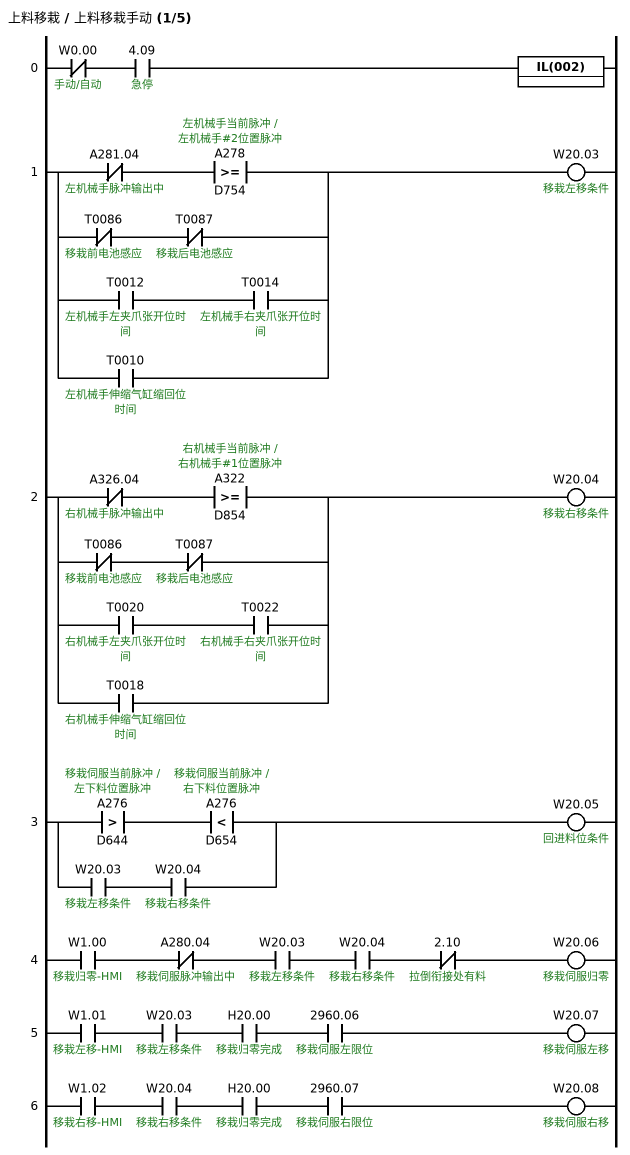
; [picture p89: 上料移栽 / 上料移栽手动, rungs 0-6]
; rung 0
LDNOT W0.00  ; 手动/自动
AND 4.09  ; 急停
IL(002)
; rung 1
LDNOT A281.04  ; 左机械手脉冲输出中
AND>=SL(328) A278 D754  ; 左机械手当前脉冲, 左机械手#2位置脉冲
LDNOT T0086  ; 移栽前电池感应
ANDNOT T0087  ; 移栽后电池感应
ORLD
LD T0012  ; 左机械手左夹爪张开位时间
AND T0014  ; 左机械手右夹爪张开位时间
ORLD
OR T0010  ; 左机械手伸缩气缸缩回位时间
OUT W20.03  ; 移栽左移条件
; rung 2
LDNOT A326.04  ; 右机械手脉冲输出中
AND>=SL(328) A322 D854  ; 右机械手当前脉冲, 右机械手#1位置脉冲
LDNOT T0086  ; 移栽前电池感应
ANDNOT T0087  ; 移栽后电池感应
ORLD
LD T0020  ; 右机械手左夹爪张开位时间
AND T0022  ; 右机械手右夹爪张开位时间
ORLD
OR T0018  ; 右机械手伸缩气缸缩回位时间
OUT W20.04  ; 移栽右移条件
; rung 3
LD>SL(323) A276 D644  ; 移栽伺服当前脉冲, 左下料位置脉冲
AND<SL(313) A276 D654  ; 移栽伺服当前脉冲, 右下料位置脉冲
LD W20.03  ; 移栽左移条件
AND W20.04  ; 移栽右移条件
ORLD
OUT W20.05  ; 回进料位条件
; rung 4
LD W1.00  ; 移栽归零-HMI
ANDNOT A280.04  ; 移栽伺服脉冲输出中
AND W20.03  ; 移栽左移条件
AND W20.04  ; 移栽右移条件
ANDNOT 2.10  ; 拉倒衔接处有料
OUT W20.06  ; 移栽伺服归零
; rung 5
LD W1.01  ; 移栽左移-HMI
AND W20.03  ; 移栽左移条件
AND H20.00  ; 移栽归零完成
AND 2960.06  ; 移栽伺服左限位
OUT W20.07  ; 移栽伺服左移
; rung 6
LD W1.02  ; 移栽右移-HMI
AND W20.04  ; 移栽右移条件
AND H20.00  ; 移栽归零完成
AND 2960.07  ; 移栽伺服右限位
OUT W20.08  ; 移栽伺服右移

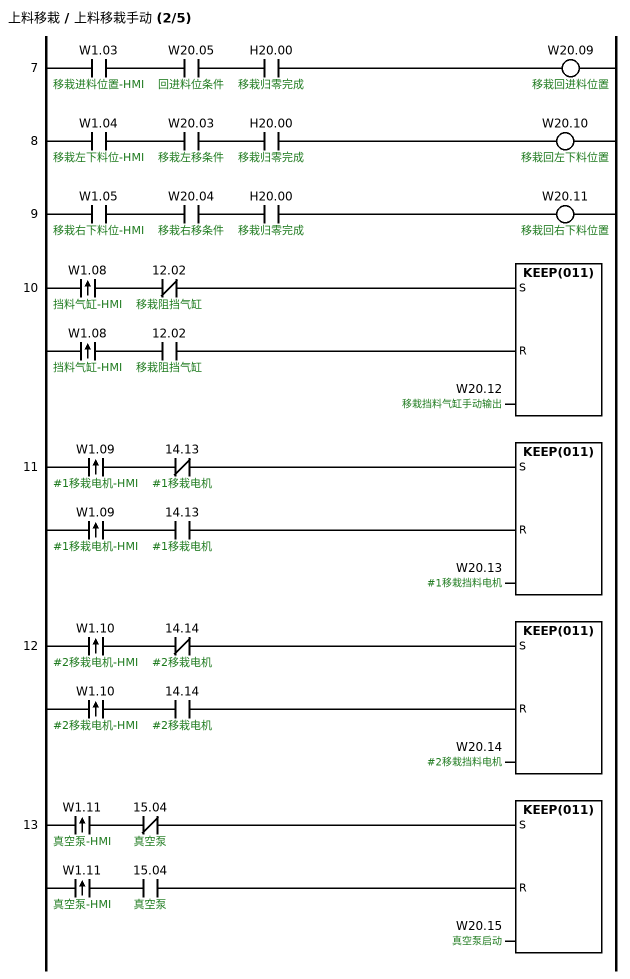
; rung 7
LD W1.03  ; 移栽进料位置-HMI
AND W20.05  ; 回进料位条件
AND H20.00  ; 移栽归零完成
OUT W20.09  ; 移栽回进料位置
; rung 8
LD W1.04  ; 移栽左下料位-HMI
AND W20.03  ; 移栽左移条件
AND H20.00  ; 移栽归零完成
OUT W20.10  ; 移栽回左下料位置
; rung 9
LD W1.05  ; 移栽右下料位-HMI
AND W20.04  ; 移栽右移条件
AND H20.00  ; 移栽归零完成
OUT W20.11  ; 移栽回右下料位置
; rung 10
@LD W1.08  ; 挡料气缸-HMI
ANDNOT 12.02  ; 移栽阻挡气缸
@LD W1.08  ; 挡料气缸-HMI
AND 12.02  ; 移栽阻挡气缸
KEEP(011) W20.12  ; 移栽挡料气缸手动输出
; rung 11
@LD W1.09  ; #1移栽电机-HMI
ANDNOT 14.13  ; #1移栽电机
@LD W1.09  ; #1移栽电机-HMI
AND 14.13  ; #1移栽电机
KEEP(011) W20.13  ; #1移栽挡料电机
; rung 12
@LD W1.10  ; #2移栽电机-HMI
ANDNOT 14.14  ; #2移栽电机
@LD W1.10  ; #2移栽电机-HMI
AND 14.14  ; #2移栽电机
KEEP(011) W20.14  ; #2移栽挡料电机
; rung 13
@LD W1.11  ; 真空泵-HMI
ANDNOT 15.04  ; 真空泵
@LD W1.11  ; 真空泵-HMI
AND 15.04  ; 真空泵
KEEP(011) W20.15  ; 真空泵启动

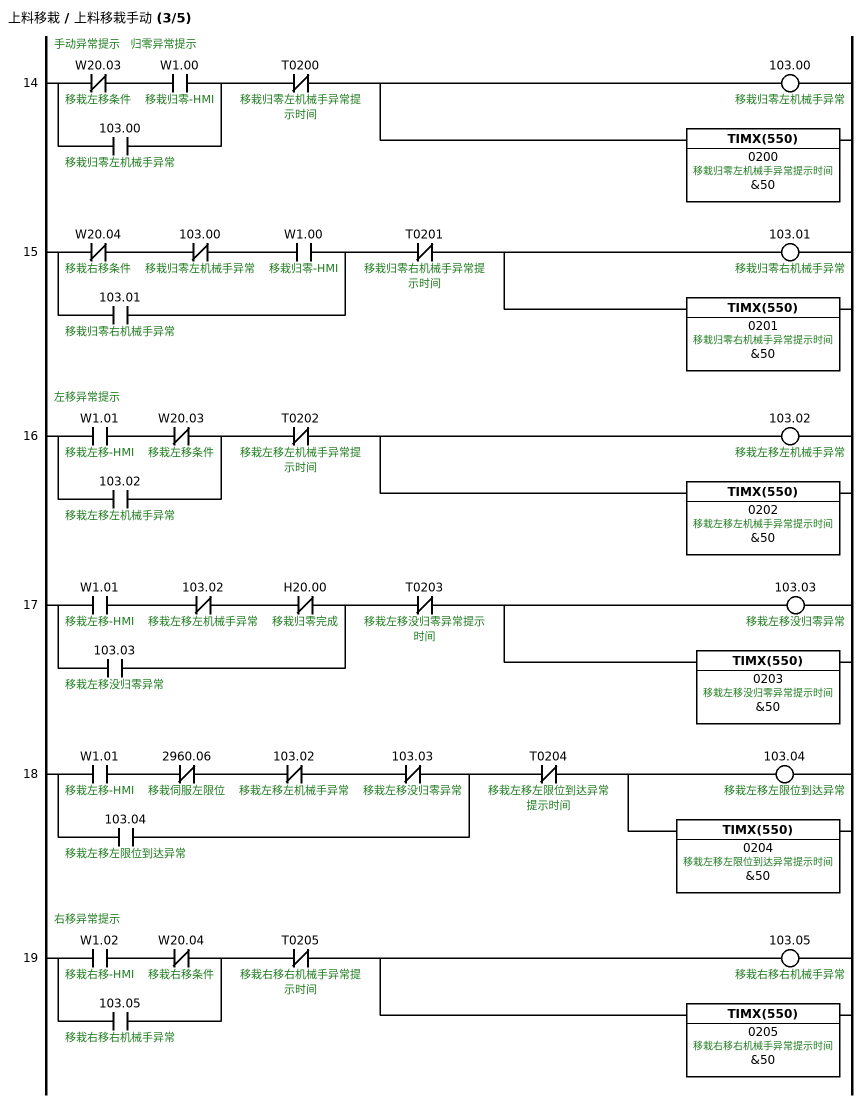
; rung 14: 手动异常提示   归零异常提示
LDNOT W20.03  ; 移栽左移条件
AND W1.00  ; 移栽归零-HMI
OR 103.00  ; 移栽归零左机械手异常
ANDNOT T0200  ; 移栽归零左机械手异常提示时间
OUT 103.00  ; 移栽归零左机械手异常
TIMX(550) 0200 &50  ; 移栽归零左机械手异常提示时间
; rung 15
LDNOT W20.04  ; 移栽右移条件
ANDNOT 103.00  ; 移栽归零左机械手异常
AND W1.00  ; 移栽归零-HMI
OR 103.01  ; 移栽归零右机械手异常
ANDNOT T0201  ; 移栽归零右机械手异常提示时间
OUT 103.01  ; 移栽归零右机械手异常
TIMX(550) 0201 &50  ; 移栽归零右机械手异常提示时间
; rung 16: 左移异常提示
LD W1.01  ; 移栽左移-HMI
ANDNOT W20.03  ; 移栽左移条件
OR 103.02  ; 移栽左移左机械手异常
ANDNOT T0202  ; 移栽左移左机械手异常提示时间
OUT 103.02  ; 移栽左移左机械手异常
TIMX(550) 0202 &50  ; 移栽左移左机械手异常提示时间
; rung 17
LD W1.01  ; 移栽左移-HMI
ANDNOT 103.02  ; 移栽左移左机械手异常
ANDNOT H20.00  ; 移栽归零完成
OR 103.03  ; 移栽左移没归零异常
ANDNOT T0203  ; 移栽左移没归零异常提示时间
OUT 103.03  ; 移栽左移没归零异常
TIMX(550) 0203 &50  ; 移栽左移没归零异常提示时间
; rung 18
LD W1.01  ; 移栽左移-HMI
ANDNOT 2960.06  ; 移栽伺服左限位
ANDNOT 103.02  ; 移栽左移左机械手异常
ANDNOT 103.03  ; 移栽左移没归零异常
OR 103.04  ; 移栽左移左限位到达异常
ANDNOT T0204  ; 移栽左移左限位到达异常提示时间
OUT 103.04  ; 移栽左移左限位到达异常
TIMX(550) 0204 &50  ; 移栽左移左限位到达异常提示时间
; rung 19: 右移异常提示
LD W1.02  ; 移栽右移-HMI
ANDNOT W20.04  ; 移栽右移条件
OR 103.05  ; 移栽右移右机械手异常
ANDNOT T0205  ; 移栽右移右机械手异常提示时间
OUT 103.05  ; 移栽右移右机械手异常
TIMX(550) 0205 &50  ; 移栽右移右机械手异常提示时间

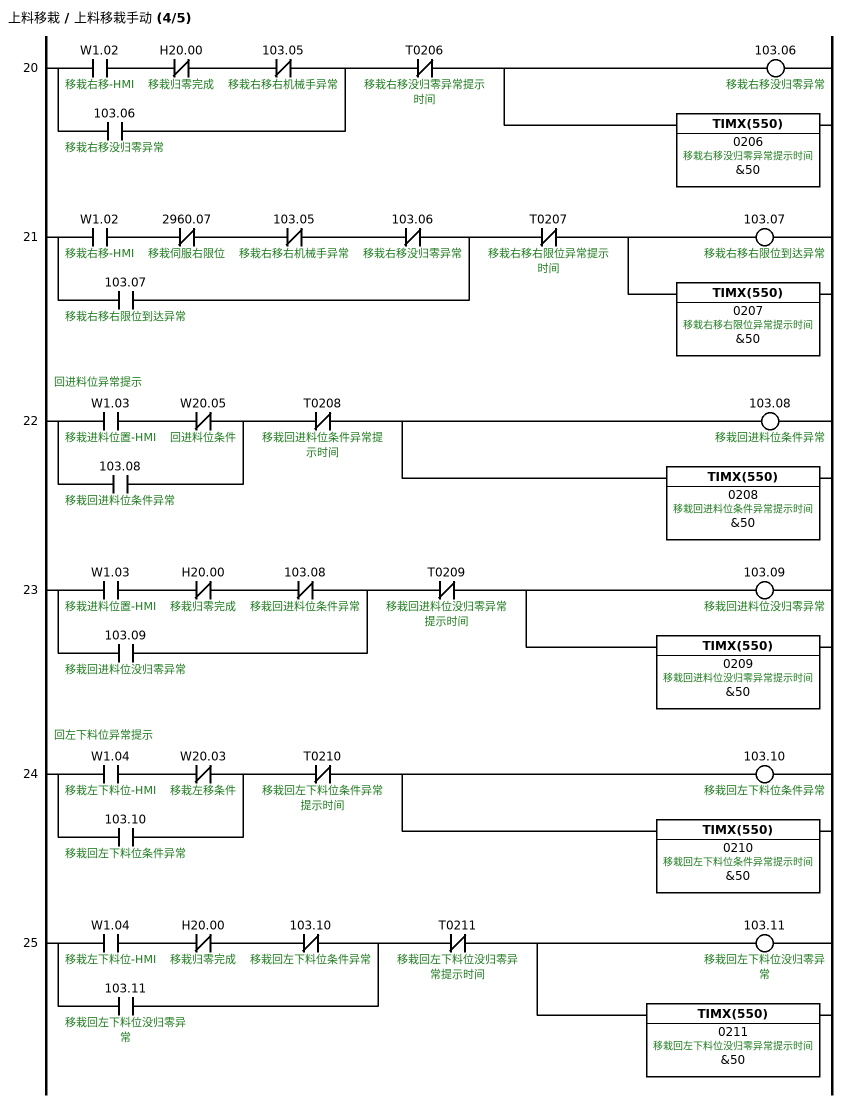
; rung 20
LD W1.02  ; 移栽右移-HMI
ANDNOT H20.00  ; 移栽归零完成
ANDNOT 103.05  ; 移栽右移右机械手异常
OR 103.06  ; 移栽右移没归零异常
ANDNOT T0206  ; 移栽右移没归零异常提示时间
OUT 103.06  ; 移栽右移没归零异常
TIMX(550) 0206 &50  ; 移栽右移没归零异常提示时间
; rung 21
LD W1.02  ; 移栽右移-HMI
ANDNOT 2960.07  ; 移栽伺服右限位
ANDNOT 103.05  ; 移栽右移右机械手异常
ANDNOT 103.06  ; 移栽右移没归零异常
OR 103.07  ; 移栽右移右限位到达异常
ANDNOT T0207  ; 移栽右移右限位异常提示时间
OUT 103.07  ; 移栽右移右限位到达异常
TIMX(550) 0207 &50  ; 移栽右移右限位异常提示时间
; rung 22: 回进料位异常提示
LD W1.03  ; 移栽进料位置-HMI
ANDNOT W20.05  ; 回进料位条件
OR 103.08  ; 移栽回进料位条件异常
ANDNOT T0208  ; 移栽回进料位条件异常提示时间
OUT 103.08  ; 移栽回进料位条件异常
TIMX(550) 0208 &50  ; 移栽回进料位条件异常提示时间
; rung 23
LD W1.03  ; 移栽进料位置-HMI
ANDNOT H20.00  ; 移栽归零完成
ANDNOT 103.08  ; 移栽回进料位条件异常
OR 103.09  ; 移栽回进料位没归零异常
ANDNOT T0209  ; 移栽回进料位没归零异常提示时间
OUT 103.09  ; 移栽回进料位没归零异常
TIMX(550) 0209 &50  ; 移栽回进料位没归零异常提示时间
; rung 24: 回左下料位异常提示
LD W1.04  ; 移栽左下料位-HMI
ANDNOT W20.03  ; 移栽左移条件
OR 103.10  ; 移栽回左下料位条件异常
ANDNOT T0210  ; 移栽回左下料位条件异常提示时间
OUT 103.10  ; 移栽回左下料位条件异常
TIMX(550) 0210 &50  ; 移栽回左下料位条件异常提示时间
; rung 25
LD W1.04  ; 移栽左下料位-HMI
ANDNOT H20.00  ; 移栽归零完成
ANDNOT 103.10  ; 移栽回左下料位条件异常
OR 103.11  ; 移栽回左下料位没归零异常
ANDNOT T0211  ; 移栽回左下料位没归零异常提示时间
OUT 103.11  ; 移栽回左下料位没归零异常
TIMX(550) 0211 &50  ; 移栽回左下料位没归零异常提示时间

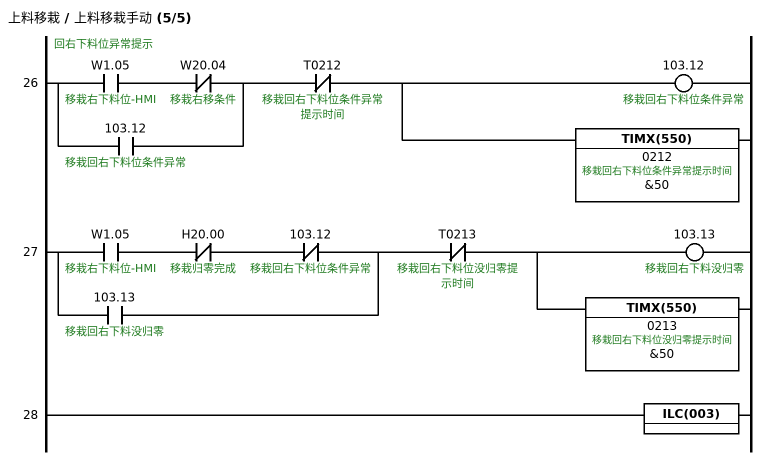
; rung 26: 回右下料位异常提示
LD W1.05  ; 移栽右下料位-HMI
ANDNOT W20.04  ; 移栽右移条件
OR 103.12  ; 移栽回右下料位条件异常
ANDNOT T0212  ; 移栽回右下料位条件异常提示时间
OUT 103.12  ; 移栽回右下料位条件异常
TIMX(550) 0212 &50  ; 移栽回右下料位条件异常提示时间
; rung 27
LD W1.05  ; 移栽右下料位-HMI
ANDNOT H20.00  ; 移栽归零完成
ANDNOT 103.12  ; 移栽回右下料位条件异常
OR 103.13  ; 移栽回右下料没归零
ANDNOT T0213  ; 移栽回右下料位没归零提示时间
OUT 103.13  ; 移栽回右下料没归零
TIMX(550) 0213 &50  ; 移栽回右下料位没归零提示时间
; rung 28
ILC(003)

### Section 上料移栽自动

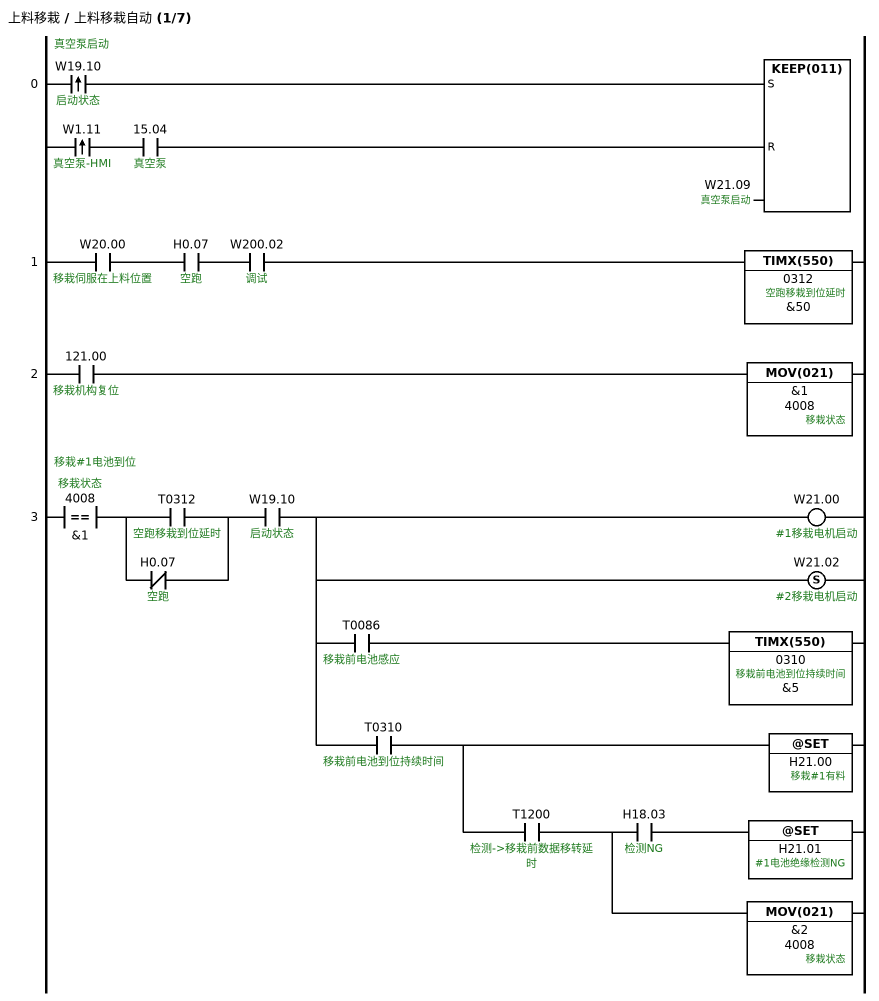
; rung 0: 真空泵启动
@LD W19.10  ; 启动状态
@LD W1.11  ; 真空泵-HMI
AND 15.04  ; 真空泵
KEEP(011) W21.09  ; 真空泵启动
; rung 1
LD W20.00  ; 移栽伺服在上料位置
AND H0.07  ; 空跑
AND W200.02  ; 调试
TIMX(550) 0312 &50  ; 空跑移栽到位延时
; rung 2
LD 121.00  ; 移栽机构复位
MOV(021) &1 4008  ; 移栽状态
; rung 3: 移栽#1电池到位
LD=(300) 4008 &1  ; 移栽状态
LD T0312  ; 空跑移栽到位延时
ORNOT H0.07  ; 空跑
ANDLD
AND W19.10  ; 启动状态
OUT TR0
OUT W21.00  ; #1移栽电机启动
SET W21.02  ; #2移栽电机启动
AND T0086  ; 移栽前电池感应
TIMX(550) 0310 &5  ; 移栽前电池到位持续时间
LD TR0
AND T0310  ; 移栽前电池到位持续时间
@SET H21.00  ; 移栽#1有料
AND T1200  ; 检测->移栽前数据移转延时
OUT TR0
AND H18.03  ; 检测NG
@SET H21.01  ; #1电池绝缘检测NG
LD TR0
MOV(021) &2 4008  ; 移栽状态

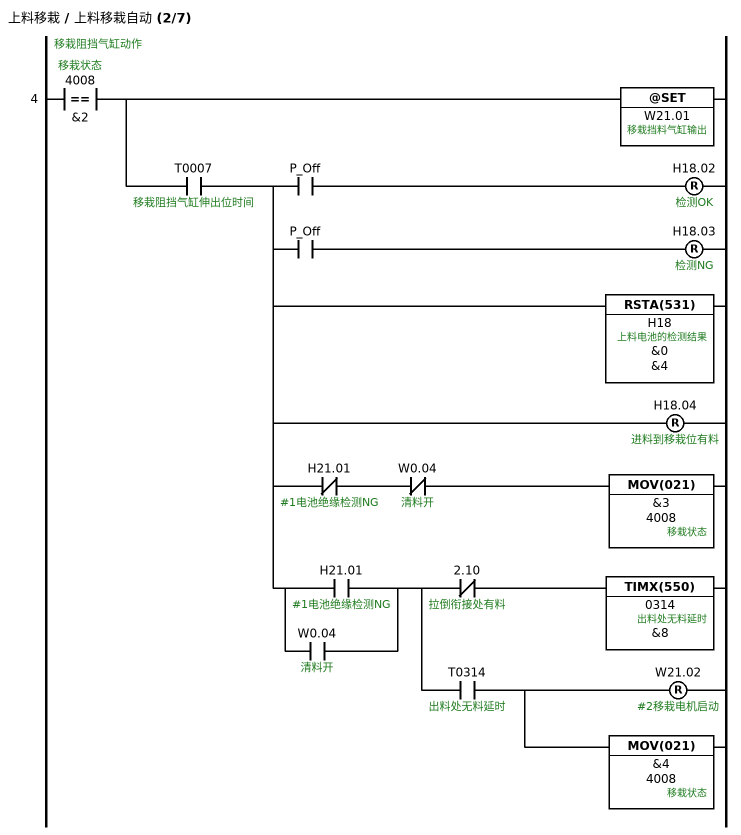
; rung 4: 移栽阻挡气缸动作
LD=(300) 4008 &2  ; 移栽状态
@SET W21.01  ; 移栽挡料气缸输出
AND T0007  ; 移栽阻挡气缸伸出位时间
OUT TR0
AND P_Off
RSET H18.02  ; 检测OK
LD TR0
AND P_Off
RSET H18.03  ; 检测NG
LD TR0
RSTA(531) H18 &0 &4  ; 上料电池的检测结果
RSET H18.04  ; 进料到移栽位有料
ANDNOT H21.01  ; #1电池绝缘检测NG
ANDNOT W0.04  ; 清料开
MOV(021) &3 4008  ; 移栽状态
LD TR0
LD H21.01  ; #1电池绝缘检测NG
OR W0.04  ; 清料开
ANDLD
OUT TR0
ANDNOT 2.10  ; 拉倒衔接处有料
TIMX(550) 0314 &8  ; 出料处无料延时
LD TR0
AND T0314  ; 出料处无料延时
RSET W21.02  ; #2移栽电机启动
MOV(021) &4 4008  ; 移栽状态

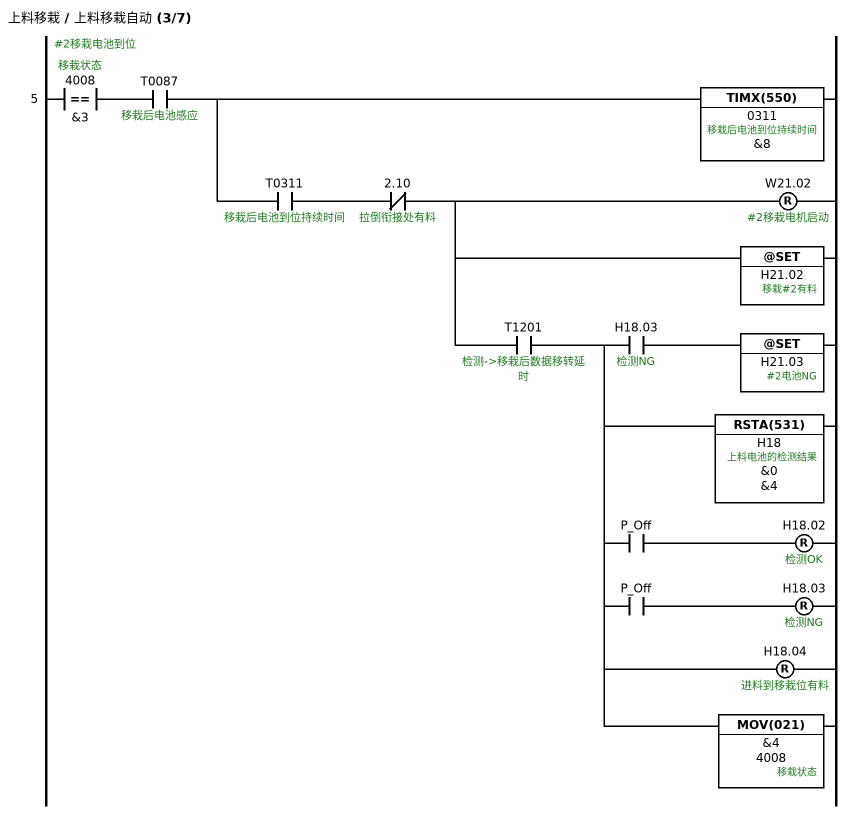
; rung 5: #2移栽电池到位
LD=(300) 4008 &3  ; 移栽状态
AND T0087  ; 移栽后电池感应
TIMX(550) 0311 &8  ; 移栽后电池到位持续时间
AND T0311  ; 移栽后电池到位持续时间
ANDNOT 2.10  ; 拉倒衔接处有料
RSET W21.02  ; #2移栽电机启动
@SET H21.02  ; 移栽#2有料
AND T1201  ; 检测->移栽后数据移转延时
OUT TR0
AND H18.03  ; 检测NG
@SET H21.03  ; #2电池NG
LD TR0
RSTA(531) H18 &0 &4  ; 上料电池的检测结果
AND P_Off
RSET H18.02  ; 检测OK
LD TR0
AND P_Off
RSET H18.03  ; 检测NG
LD TR0
RSET H18.04  ; 进料到移栽位有料
MOV(021) &4 4008  ; 移栽状态

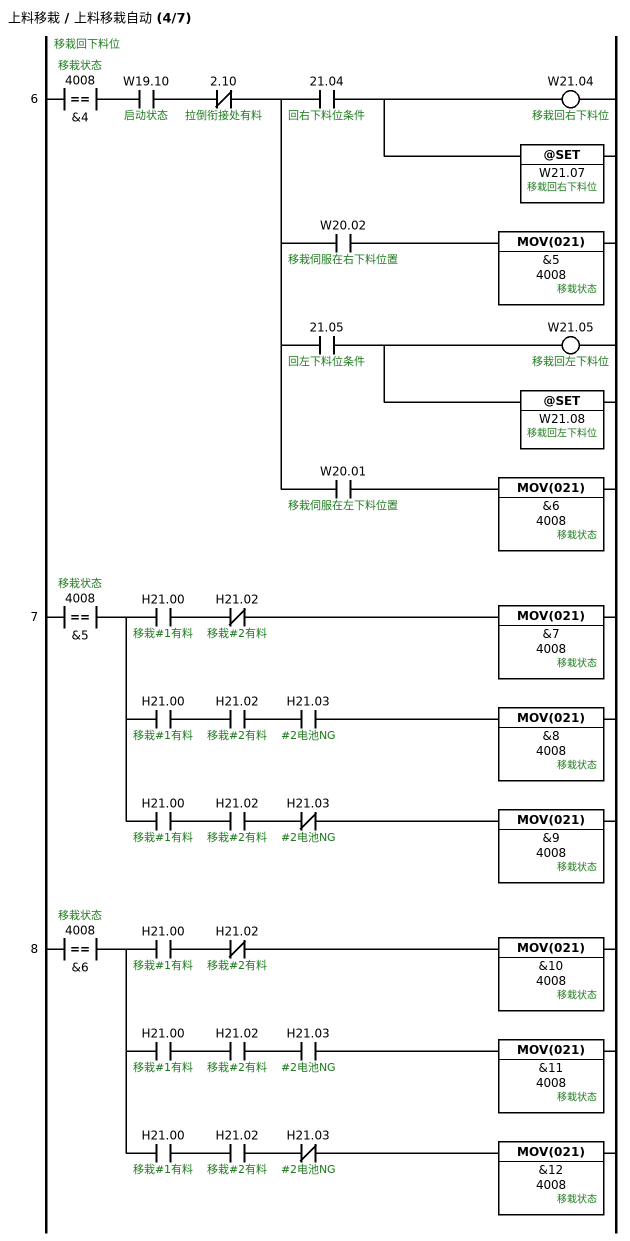
; rung 6: 移栽回下料位
LD=(300) 4008 &4  ; 移栽状态
AND W19.10  ; 启动状态
ANDNOT 2.10  ; 拉倒衔接处有料
OUT TR0
AND 21.04  ; 回右下料位条件
OUT W21.04  ; 移栽回右下料位
@SET W21.07  ; 移栽回右下料位
LD TR0
AND W20.02  ; 移栽伺服在右下料位置
MOV(021) &5 4008  ; 移栽状态
LD TR0
AND 21.05  ; 回左下料位条件
OUT W21.05  ; 移栽回左下料位
@SET W21.08  ; 移栽回左下料位
LD TR0
AND W20.01  ; 移栽伺服在左下料位置
MOV(021) &6 4008  ; 移栽状态
; rung 7
LD=(300) 4008 &5  ; 移栽状态
OUT TR0
AND H21.00  ; 移栽#1有料
ANDNOT H21.02  ; 移栽#2有料
MOV(021) &7 4008  ; 移栽状态
LD TR0
AND H21.00  ; 移栽#1有料
AND H21.02  ; 移栽#2有料
AND H21.03  ; #2电池NG
MOV(021) &8 4008  ; 移栽状态
LD TR0
AND H21.00  ; 移栽#1有料
AND H21.02  ; 移栽#2有料
ANDNOT H21.03  ; #2电池NG
MOV(021) &9 4008  ; 移栽状态
; rung 8
LD=(300) 4008 &6  ; 移栽状态
OUT TR0
AND H21.00  ; 移栽#1有料
ANDNOT H21.02  ; 移栽#2有料
MOV(021) &10 4008  ; 移栽状态
LD TR0
AND H21.00  ; 移栽#1有料
AND H21.02  ; 移栽#2有料
AND H21.03  ; #2电池NG
MOV(021) &11 4008  ; 移栽状态
LD TR0
AND H21.00  ; 移栽#1有料
AND H21.02  ; 移栽#2有料
ANDNOT H21.03  ; #2电池NG
MOV(021) &12 4008  ; 移栽状态

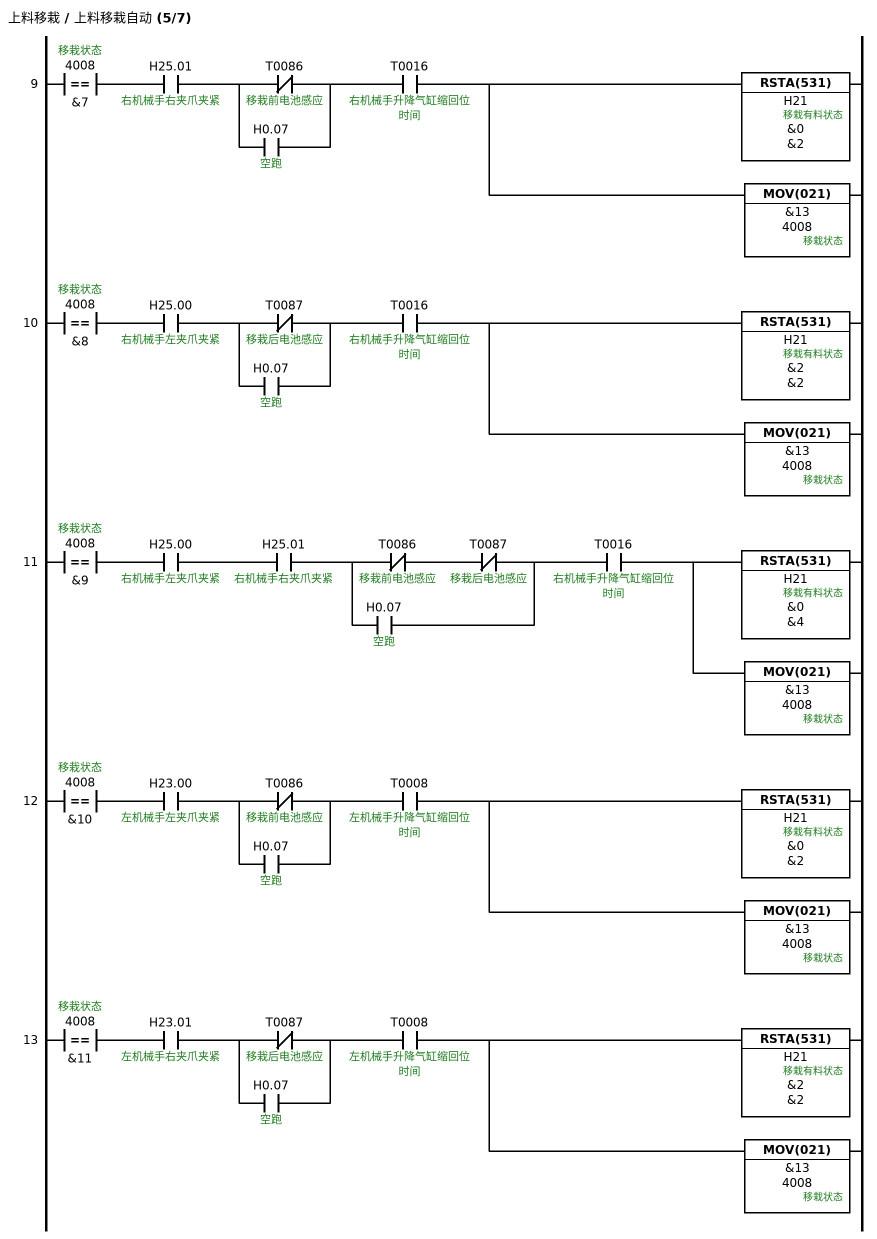
; rung 9
LD=(300) 4008 &7  ; 移栽状态
AND H25.01  ; 右机械手右夹爪夹紧
LDNOT T0086  ; 移栽前电池感应
OR H0.07  ; 空跑
ANDLD
AND T0016  ; 右机械手升降气缸缩回位时间
RSTA(531) H21 &0 &2  ; 移栽有料状态
MOV(021) &13 4008  ; 移栽状态
; rung 10
LD=(300) 4008 &8  ; 移栽状态
AND H25.00  ; 右机械手左夹爪夹紧
LDNOT T0087  ; 移栽后电池感应
OR H0.07  ; 空跑
ANDLD
AND T0016  ; 右机械手升降气缸缩回位时间
RSTA(531) H21 &2 &2  ; 移栽有料状态
MOV(021) &13 4008  ; 移栽状态
; rung 11
LD=(300) 4008 &9  ; 移栽状态
AND H25.00  ; 右机械手左夹爪夹紧
AND H25.01  ; 右机械手右夹爪夹紧
LDNOT T0086  ; 移栽前电池感应
ANDNOT T0087  ; 移栽后电池感应
OR H0.07  ; 空跑
ANDLD
AND T0016  ; 右机械手升降气缸缩回位时间
RSTA(531) H21 &0 &4  ; 移栽有料状态
MOV(021) &13 4008  ; 移栽状态
; rung 12
LD=(300) 4008 &10  ; 移栽状态
AND H23.00  ; 左机械手左夹爪夹紧
LDNOT T0086  ; 移栽前电池感应
OR H0.07  ; 空跑
ANDLD
AND T0008  ; 左机械手升降气缸缩回位时间
RSTA(531) H21 &0 &2  ; 移栽有料状态
MOV(021) &13 4008  ; 移栽状态
; rung 13
LD=(300) 4008 &11  ; 移栽状态
AND H23.01  ; 左机械手右夹爪夹紧
LDNOT T0087  ; 移栽后电池感应
OR H0.07  ; 空跑
ANDLD
AND T0008  ; 左机械手升降气缸缩回位时间
RSTA(531) H21 &2 &2  ; 移栽有料状态
MOV(021) &13 4008  ; 移栽状态

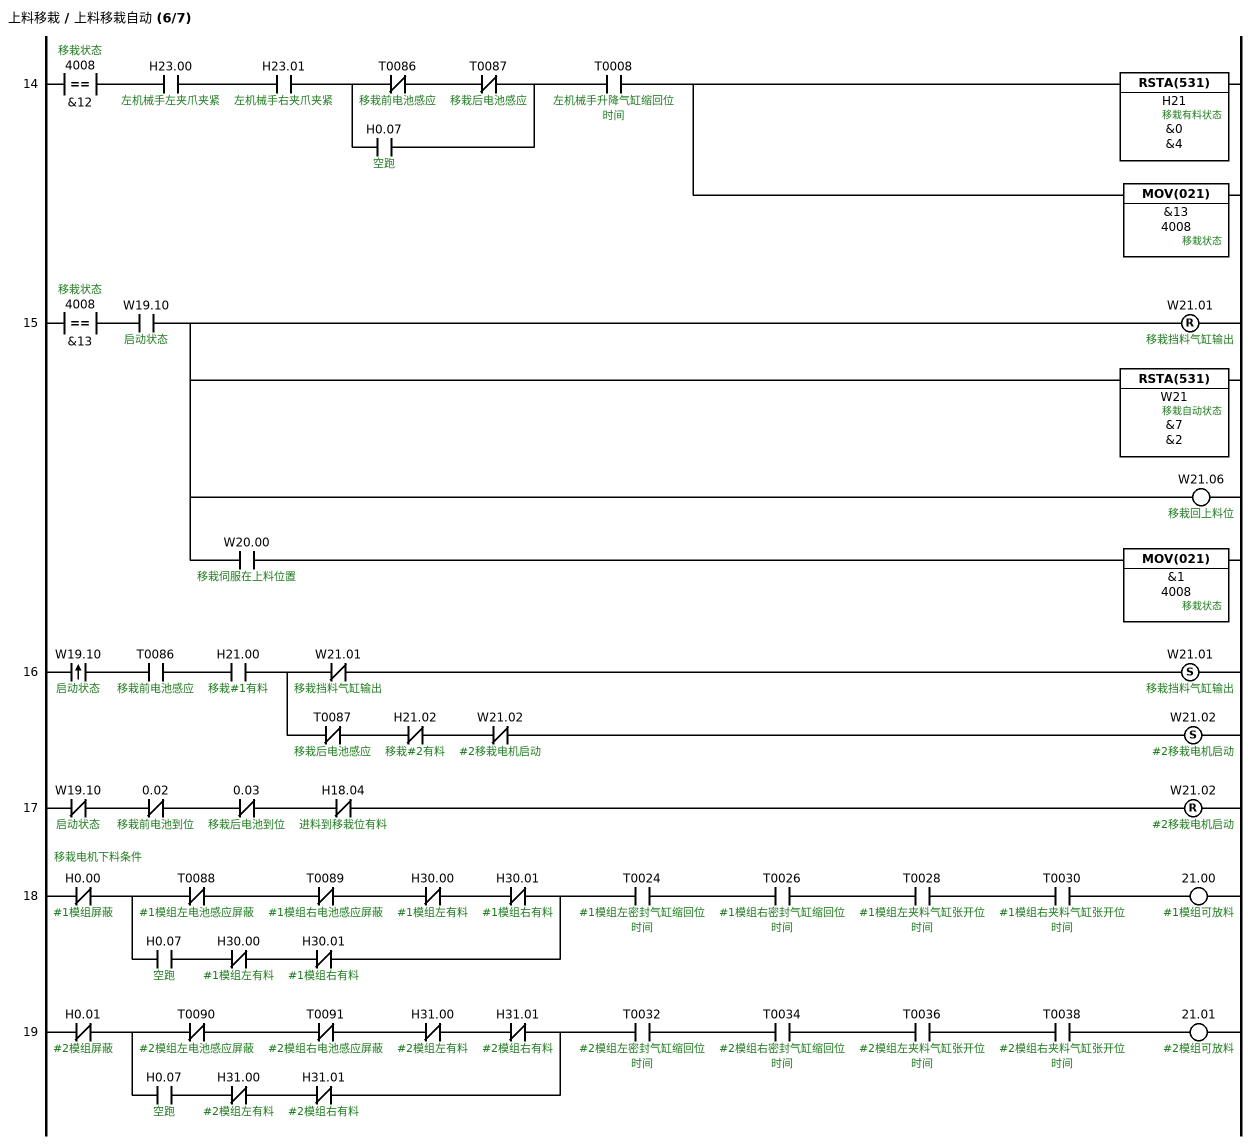
; rung 14
LD=(300) 4008 &12  ; 移栽状态
AND H23.00  ; 左机械手左夹爪夹紧
AND H23.01  ; 左机械手右夹爪夹紧
LDNOT T0086  ; 移栽前电池感应
ANDNOT T0087  ; 移栽后电池感应
OR H0.07  ; 空跑
ANDLD
AND T0008  ; 左机械手升降气缸缩回位时间
RSTA(531) H21 &0 &4  ; 移栽有料状态
MOV(021) &13 4008  ; 移栽状态
; rung 15
LD=(300) 4008 &13  ; 移栽状态
AND W19.10  ; 启动状态
RSET W21.01  ; 移栽挡料气缸输出
RSTA(531) W21 &7 &2  ; 移栽自动状态
OUT W21.06  ; 移栽回上料位
AND W20.00  ; 移栽伺服在上料位置
MOV(021) &1 4008  ; 移栽状态
; rung 16
@LD W19.10  ; 启动状态
AND T0086  ; 移栽前电池感应
AND H21.00  ; 移栽#1有料
OUT TR0
ANDNOT W21.01  ; 移栽挡料气缸输出
SET W21.01  ; 移栽挡料气缸输出
LD TR0
ANDNOT T0087  ; 移栽后电池感应
ANDNOT H21.02  ; 移栽#2有料
ANDNOT W21.02  ; #2移栽电机启动
SET W21.02  ; #2移栽电机启动
; rung 17
LDNOT W19.10  ; 启动状态
ANDNOT 0.02  ; 移栽前电池到位
ANDNOT 0.03  ; 移栽后电池到位
ANDNOT H18.04  ; 进料到移栽位有料
RSET W21.02  ; #2移栽电机启动
; rung 18: 移栽电机下料条件
LDNOT H0.00  ; #1模组屏蔽
LDNOT T0088  ; #1模组左电池感应屏蔽
ANDNOT T0089  ; #1模组右电池感应屏蔽
ANDNOT H30.00  ; #1模组左有料
ANDNOT H30.01  ; #1模组右有料
LD H0.07  ; 空跑
ANDNOT H30.00  ; #1模组左有料
ANDNOT H30.01  ; #1模组右有料
ORLD
ANDLD
AND T0024  ; #1模组左密封气缸缩回位时间
AND T0026  ; #1模组右密封气缸缩回位时间
AND T0028  ; #1模组左夹料气缸张开位时间
AND T0030  ; #1模组右夹料气缸张开位时间
OUT 21.00  ; #1模组可放料
; rung 19
LDNOT H0.01  ; #2模组屏蔽
LDNOT T0090  ; #2模组左电池感应屏蔽
ANDNOT T0091  ; #2模组右电池感应屏蔽
ANDNOT H31.00  ; #2模组左有料
ANDNOT H31.01  ; #2模组右有料
LD H0.07  ; 空跑
ANDNOT H31.00  ; #2模组左有料
ANDNOT H31.01  ; #2模组右有料
ORLD
ANDLD
AND T0032  ; #2模组左密封气缸缩回位时间
AND T0034  ; #2模组右密封气缸缩回位时间
AND T0036  ; #2模组左夹料气缸张开位时间
AND T0038  ; #2模组右夹料气缸张开位时间
OUT 21.01  ; #2模组可放料

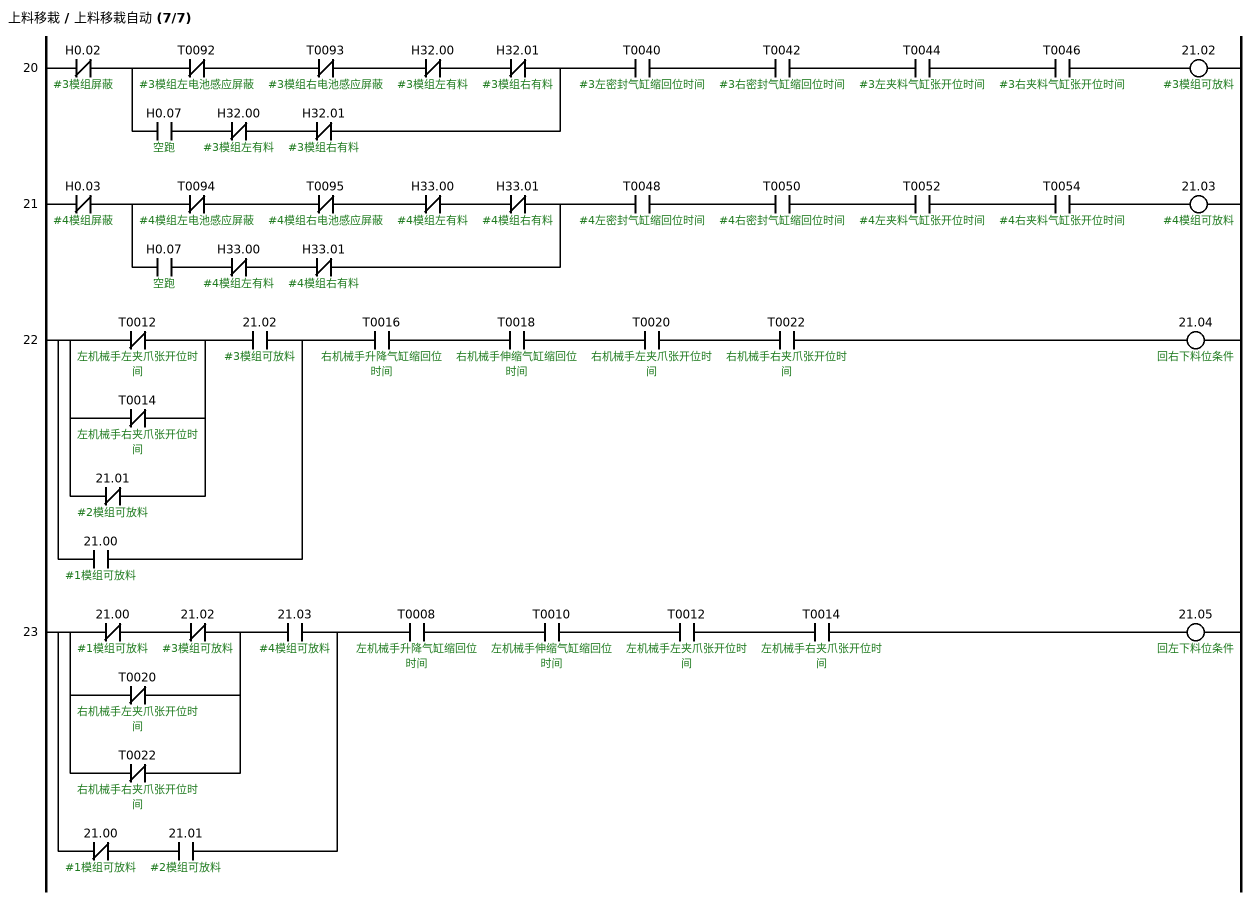
; rung 20
LDNOT H0.02  ; #3模组屏蔽
LDNOT T0092  ; #3模组左电池感应屏蔽
ANDNOT T0093  ; #3模组右电池感应屏蔽
ANDNOT H32.00  ; #3模组左有料
ANDNOT H32.01  ; #3模组右有料
LD H0.07  ; 空跑
ANDNOT H32.00  ; #3模组左有料
ANDNOT H32.01  ; #3模组右有料
ORLD
ANDLD
AND T0040  ; #3左密封气缸缩回位时间
AND T0042  ; #3右密封气缸缩回位时间
AND T0044  ; #3左夹料气缸张开位时间
AND T0046  ; #3右夹料气缸张开位时间
OUT 21.02  ; #3模组可放料
; rung 21
LDNOT H0.03  ; #4模组屏蔽
LDNOT T0094  ; #4模组左电池感应屏蔽
ANDNOT T0095  ; #4模组右电池感应屏蔽
ANDNOT H33.00  ; #4模组左有料
ANDNOT H33.01  ; #4模组右有料
LD H0.07  ; 空跑
ANDNOT H33.00  ; #4模组左有料
ANDNOT H33.01  ; #4模组右有料
ORLD
ANDLD
AND T0048  ; #4左密封气缸缩回位时间
AND T0050  ; #4右密封气缸缩回位时间
AND T0052  ; #4左夹料气缸张开位时间
AND T0054  ; #4右夹料气缸张开位时间
OUT 21.03  ; #4模组可放料
; rung 22
LDNOT T0012  ; 左机械手左夹爪张开位时间
ORNOT T0014  ; 左机械手右夹爪张开位时间
ORNOT 21.01  ; #2模组可放料
AND 21.02  ; #3模组可放料
OR 21.00  ; #1模组可放料
AND T0016  ; 右机械手升降气缸缩回位时间
AND T0018  ; 右机械手伸缩气缸缩回位时间
AND T0020  ; 右机械手左夹爪张开位时间
AND T0022  ; 右机械手右夹爪张开位时间
OUT 21.04  ; 回右下料位条件
; rung 23
LDNOT 21.00  ; #1模组可放料
ANDNOT 21.02  ; #3模组可放料
ORNOT T0020  ; 右机械手左夹爪张开位时间
ORNOT T0022  ; 右机械手右夹爪张开位时间
AND 21.03  ; #4模组可放料
LDNOT 21.00  ; #1模组可放料
AND 21.01  ; #2模组可放料
ORLD
AND T0008  ; 左机械手升降气缸缩回位时间
AND T0010  ; 左机械手伸缩气缸缩回位时间
AND T0012  ; 左机械手左夹爪张开位时间
AND T0014  ; 左机械手右夹爪张开位时间
OUT 21.05  ; 回左下料位条件

### Section 伺服参数

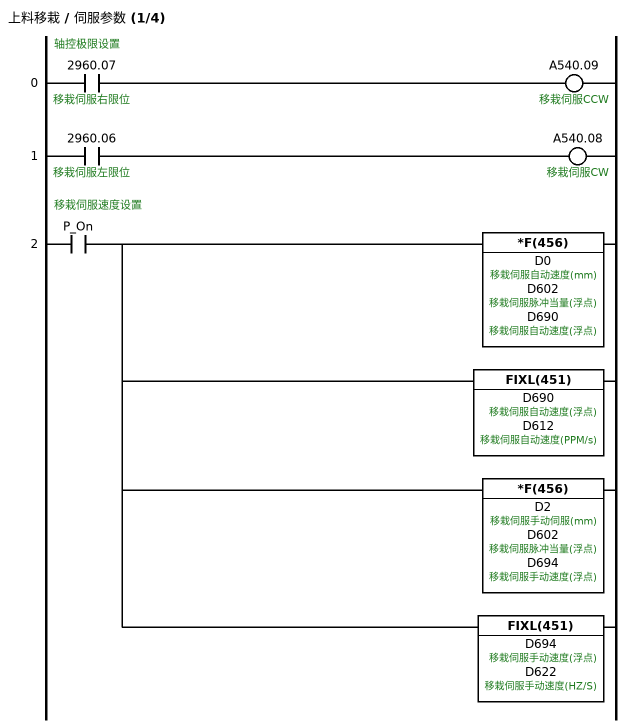
; rung 0: 轴控极限设置
LD 2960.07  ; 移栽伺服右限位
OUT A540.09  ; 移栽伺服CCW
; rung 1
LD 2960.06  ; 移栽伺服左限位
OUT A540.08  ; 移栽伺服CW
; rung 2: 移栽伺服速度设置
LD P_On
*F(456) D0 D602 D690  ; 移栽伺服自动速度(mm), 移栽伺服脉冲当量(浮点), 移栽伺服自动速度(浮点)
FIXL(451) D690 D612  ; 移栽伺服自动速度(浮点), 移栽伺服自动速度(PPM/s)
*F(456) D2 D602 D694  ; 移栽伺服手动伺服(mm), 移栽伺服脉冲当量(浮点), 移栽伺服手动速度(浮点)
FIXL(451) D694 D622  ; 移栽伺服手动速度(浮点), 移栽伺服手动速度(HZ/S)

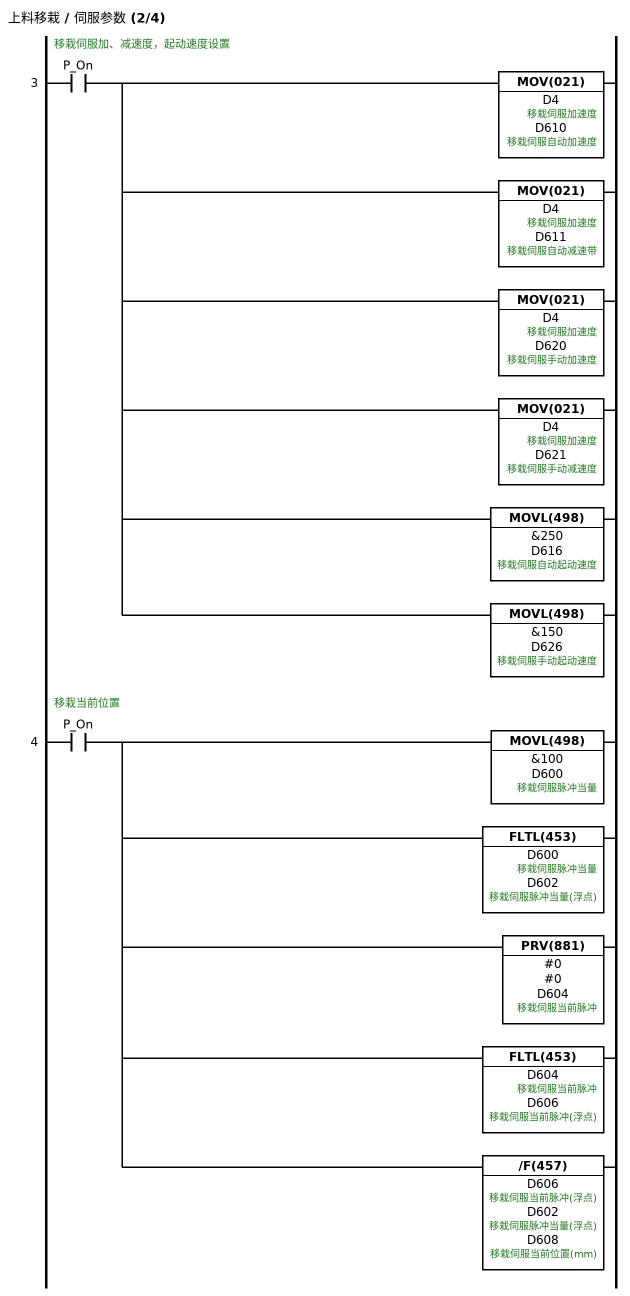
; rung 3: 移栽伺服加、减速度，起动速度设置
LD P_On
MOV(021) D4 D610  ; 移栽伺服加速度, 移栽伺服自动加速度
MOV(021) D4 D611  ; 移栽伺服加速度, 移栽伺服自动减速带
MOV(021) D4 D620  ; 移栽伺服加速度, 移栽伺服手动加速度
MOV(021) D4 D621  ; 移栽伺服加速度, 移栽伺服手动减速度
MOVL(498) &250 D616  ; 移栽伺服自动起动速度
MOVL(498) &150 D626  ; 移栽伺服手动起动速度
; rung 4: 移栽当前位置
LD P_On
MOVL(498) &100 D600  ; 移栽伺服脉冲当量
FLTL(453) D600 D602  ; 移栽伺服脉冲当量, 移栽伺服脉冲当量(浮点)
PRV(881) #0 #0 D604  ; 移栽伺服当前脉冲
FLTL(453) D604 D606  ; 移栽伺服当前脉冲, 移栽伺服当前脉冲(浮点)
/F(457) D606 D602 D608  ; 移栽伺服当前脉冲(浮点), 移栽伺服脉冲当量(浮点), 移栽伺服当前位置(mm)

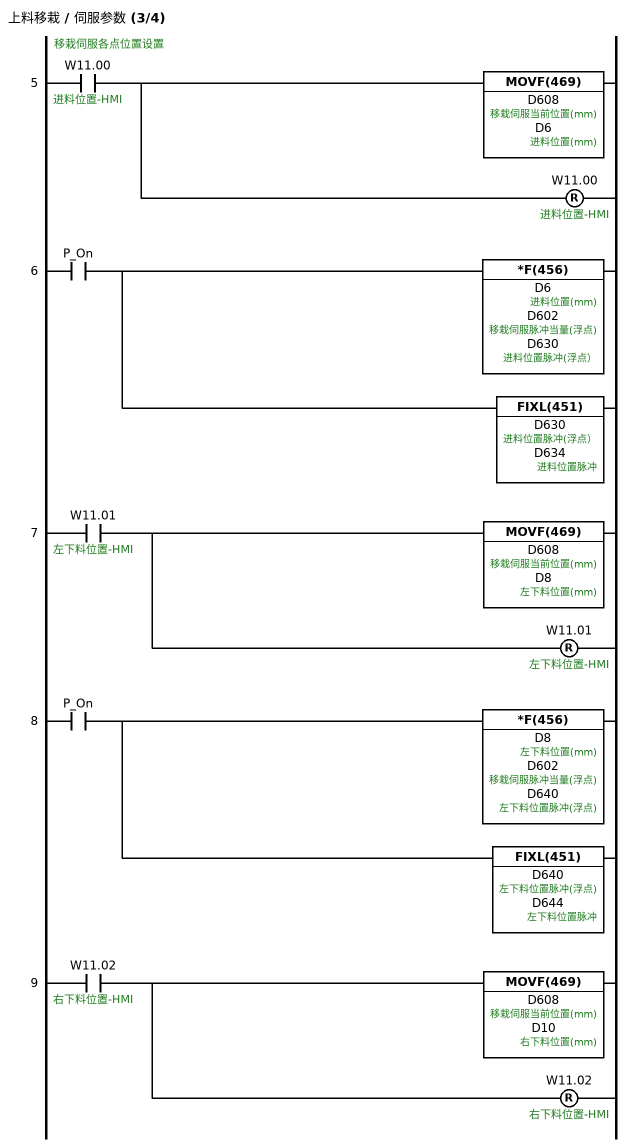
; rung 5: 移栽伺服各点位置设置
LD W11.00  ; 进料位置-HMI
MOVF(469) D608 D6  ; 移栽伺服当前位置(mm), 进料位置(mm)
RSET W11.00  ; 进料位置-HMI
; rung 6
LD P_On
*F(456) D6 D602 D630  ; 进料位置(mm), 移栽伺服脉冲当量(浮点), 进料位置脉冲(浮点）
FIXL(451) D630 D634  ; 进料位置脉冲(浮点）, 进料位置脉冲
; rung 7
LD W11.01  ; 左下料位置-HMI
MOVF(469) D608 D8  ; 移栽伺服当前位置(mm), 左下料位置(mm)
RSET W11.01  ; 左下料位置-HMI
; rung 8
LD P_On
*F(456) D8 D602 D640  ; 左下料位置(mm), 移栽伺服脉冲当量(浮点), 左下料位置脉冲(浮点)
FIXL(451) D640 D644  ; 左下料位置脉冲(浮点), 左下料位置脉冲
; rung 9
LD W11.02  ; 右下料位置-HMI
MOVF(469) D608 D10  ; 移栽伺服当前位置(mm), 右下料位置(mm)
RSET W11.02  ; 右下料位置-HMI

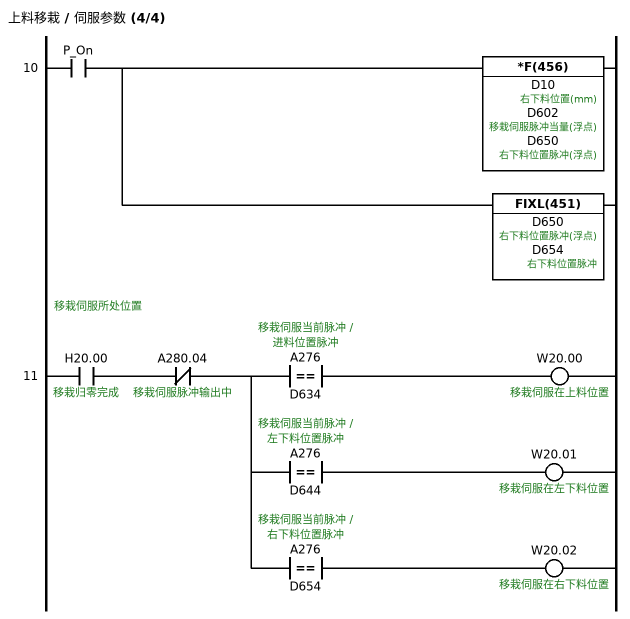
; rung 10
LD P_On
*F(456) D10 D602 D650  ; 右下料位置(mm), 移栽伺服脉冲当量(浮点), 右下料位置脉冲(浮点)
FIXL(451) D650 D654  ; 右下料位置脉冲(浮点), 右下料位置脉冲
; rung 11: 移栽伺服所处位置
LD H20.00  ; 移栽归零完成
ANDNOT A280.04  ; 移栽伺服脉冲输出中
OUT TR0
AND=SL(303) A276 D634  ; 移栽伺服当前脉冲, 进料位置脉冲
OUT W20.00  ; 移栽伺服在上料位置
LD TR0
AND=SL(303) A276 D644  ; 移栽伺服当前脉冲, 左下料位置脉冲
OUT W20.01  ; 移栽伺服在左下料位置
LD TR0
AND=SL(303) A276 D654  ; 移栽伺服当前脉冲, 右下料位置脉冲
OUT W20.02  ; 移栽伺服在右下料位置

### Section 轴控运动及外部输出

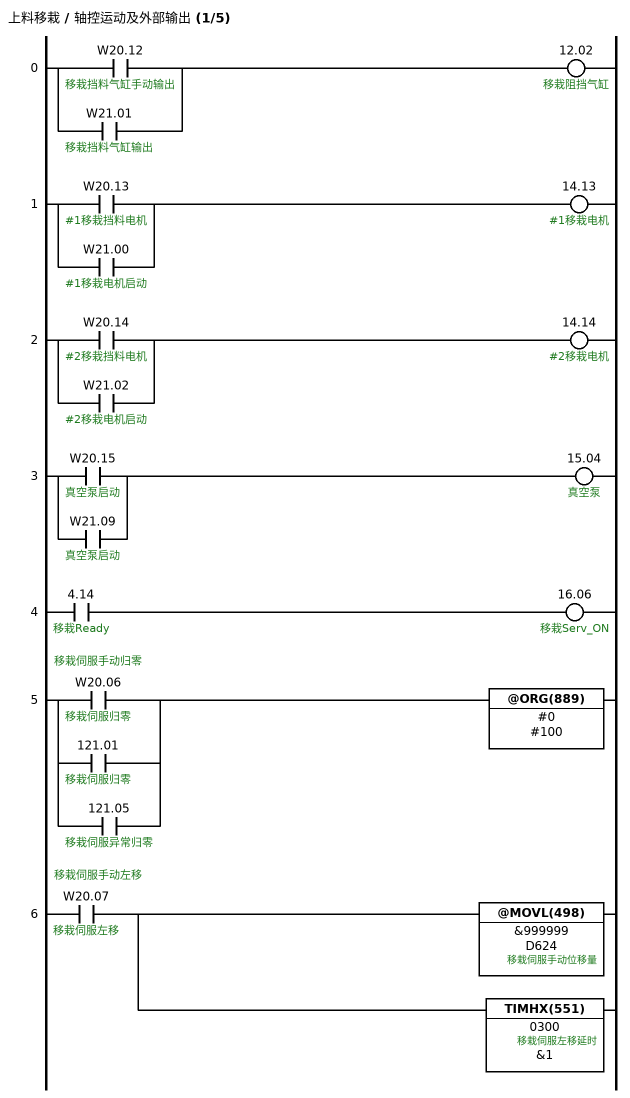
; rung 0
LD W20.12  ; 移栽挡料气缸手动输出
OR W21.01  ; 移栽挡料气缸输出
OUT 12.02  ; 移栽阻挡气缸
; rung 1
LD W20.13  ; #1移栽挡料电机
OR W21.00  ; #1移栽电机启动
OUT 14.13  ; #1移栽电机
; rung 2
LD W20.14  ; #2移栽挡料电机
OR W21.02  ; #2移栽电机启动
OUT 14.14  ; #2移栽电机
; rung 3
LD W20.15  ; 真空泵启动
OR W21.09  ; 真空泵启动
OUT 15.04  ; 真空泵
; rung 4
LD 4.14  ; 移栽Ready
OUT 16.06  ; 移栽Serv_ON
; rung 5: 移栽伺服手动归零
LD W20.06  ; 移栽伺服归零
OR 121.01  ; 移栽伺服归零
OR 121.05  ; 移栽伺服异常归零
@ORG(889) #0 #100
; rung 6: 移栽伺服手动左移
LD W20.07  ; 移栽伺服左移
@MOVL(498) &999999 D624  ; 移栽伺服手动位移量
TIMHX(551) 0300 &1  ; 移栽伺服左移延时

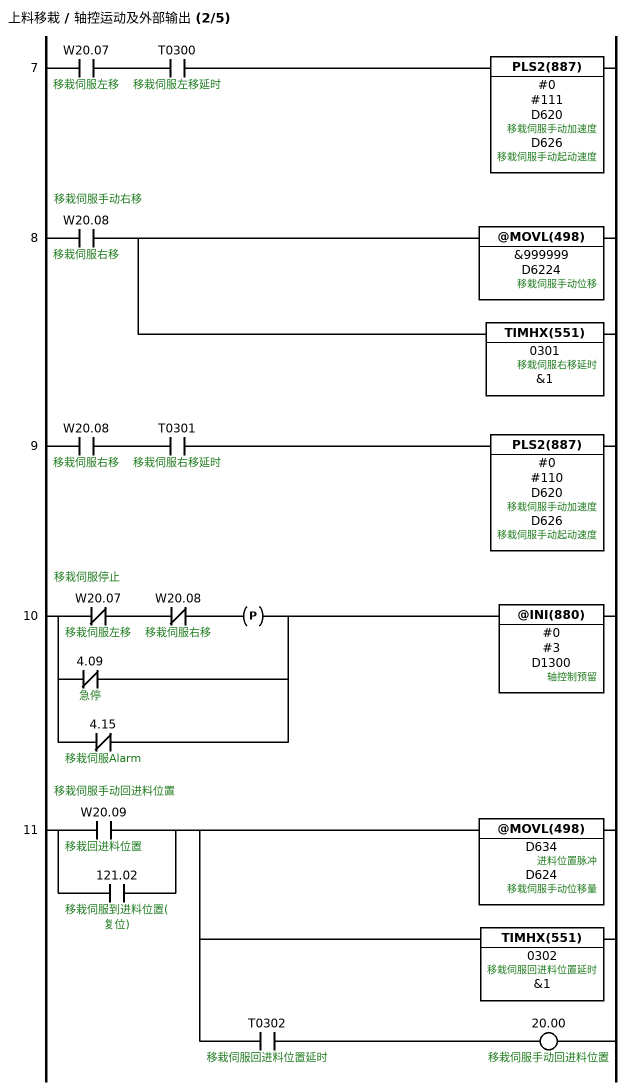
; rung 7
LD W20.07  ; 移栽伺服左移
AND T0300  ; 移栽伺服左移延时
PLS2(887) #0 #111 D620 D626  ; 移栽伺服手动加速度, 移栽伺服手动起动速度
; rung 8: 移栽伺服手动右移
LD W20.08  ; 移栽伺服右移
@MOVL(498) &999999 D6224  ; 移栽伺服手动位移
TIMHX(551) 0301 &1  ; 移栽伺服右移延时
; rung 9
LD W20.08  ; 移栽伺服右移
AND T0301  ; 移栽伺服右移延时
PLS2(887) #0 #110 D620 D626  ; 移栽伺服手动加速度, 移栽伺服手动起动速度
; rung 10: 移栽伺服停止
LDNOT W20.07  ; 移栽伺服左移
ANDNOT W20.08  ; 移栽伺服右移
UP(521)
ORNOT 4.09  ; 急停
ORNOT 4.15  ; 移栽伺服Alarm
@INI(880) #0 #3 D1300  ; 轴控制预留
; rung 11: 移栽伺服手动回进料位置
LD W20.09  ; 移栽回进料位置
OR 121.02  ; 移栽伺服到进料位置(复位)
@MOVL(498) D634 D624  ; 进料位置脉冲, 移栽伺服手动位移量
TIMHX(551) 0302 &1  ; 移栽伺服回进料位置延时
AND T0302  ; 移栽伺服回进料位置延时
OUT 20.00  ; 移栽伺服手动回进料位置

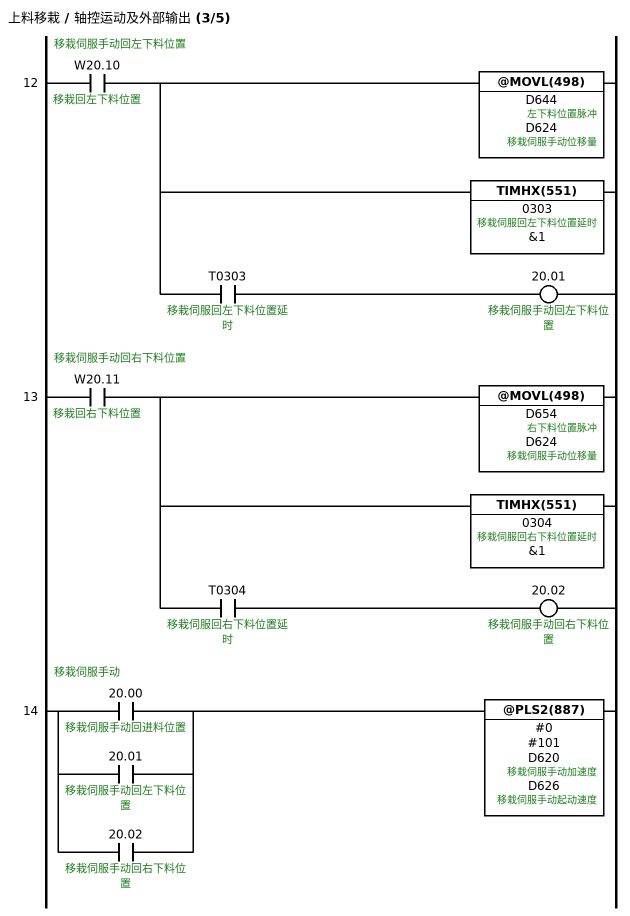
; rung 12: 移栽伺服手动回左下料位置
LD W20.10  ; 移栽回左下料位置
@MOVL(498) D644 D624  ; 左下料位置脉冲, 移栽伺服手动位移量
TIMHX(551) 0303 &1  ; 移栽伺服回左下料位置延时
AND T0303  ; 移栽伺服回左下料位置延时
OUT 20.01  ; 移栽伺服手动回左下料位置
; rung 13: 移栽伺服手动回右下料位置
LD W20.11  ; 移栽回右下料位置
@MOVL(498) D654 D624  ; 右下料位置脉冲, 移栽伺服手动位移量
TIMHX(551) 0304 &1  ; 移栽伺服回右下料位置延时
AND T0304  ; 移栽伺服回右下料位置延时
OUT 20.02  ; 移栽伺服手动回右下料位置
; rung 14: 移栽伺服手动
LD 20.00  ; 移栽伺服手动回进料位置
OR 20.01  ; 移栽伺服手动回左下料位置
OR 20.02  ; 移栽伺服手动回右下料位置
@PLS2(887) #0 #101 D620 D626  ; 移栽伺服手动加速度, 移栽伺服手动起动速度

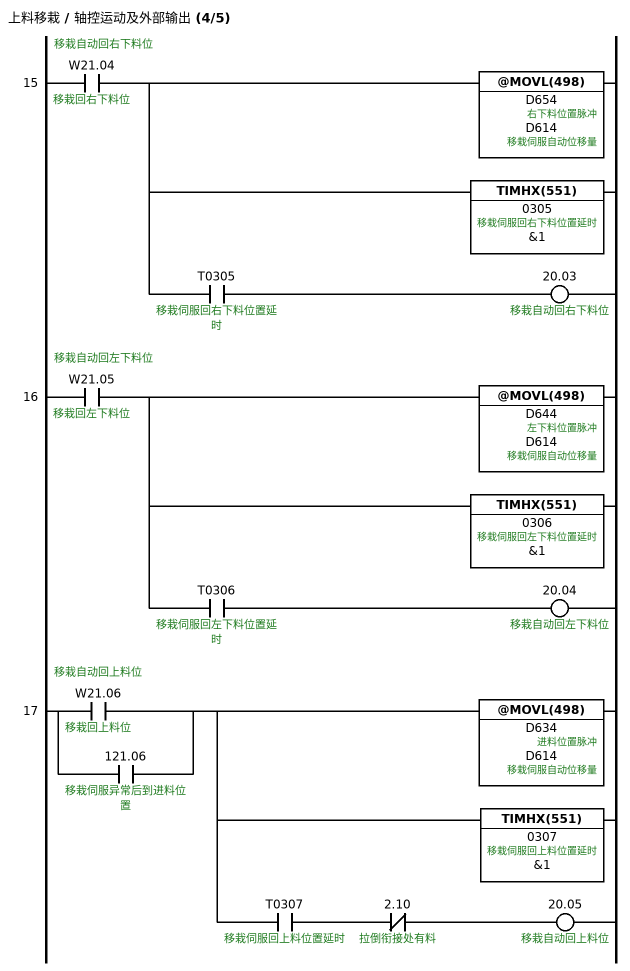
; rung 15: 移栽自动回右下料位
LD W21.04  ; 移栽回右下料位
@MOVL(498) D654 D614  ; 右下料位置脉冲, 移栽伺服自动位移量
TIMHX(551) 0305 &1  ; 移栽伺服回右下料位置延时
AND T0305  ; 移栽伺服回右下料位置延时
OUT 20.03  ; 移栽自动回右下料位
; rung 16: 移栽自动回左下料位
LD W21.05  ; 移栽回左下料位
@MOVL(498) D644 D614  ; 左下料位置脉冲, 移栽伺服自动位移量
TIMHX(551) 0306 &1  ; 移栽伺服回左下料位置延时
AND T0306  ; 移栽伺服回左下料位置延时
OUT 20.04  ; 移栽自动回左下料位
; rung 17: 移栽自动回上料位
LD W21.06  ; 移栽回上料位
OR 121.06  ; 移栽伺服异常后到进料位置
@MOVL(498) D634 D614  ; 进料位置脉冲, 移栽伺服自动位移量
TIMHX(551) 0307 &1  ; 移栽伺服回上料位置延时
AND T0307  ; 移栽伺服回上料位置延时
ANDNOT 2.10  ; 拉倒衔接处有料
OUT 20.05  ; 移栽自动回上料位

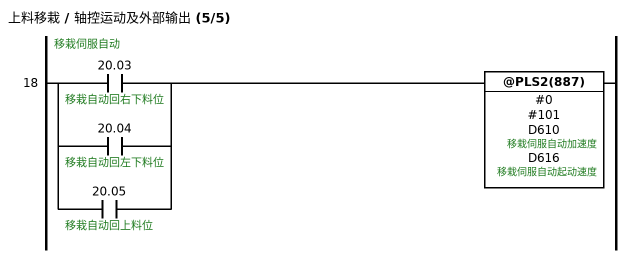
; rung 18: 移栽伺服自动
LD 20.03  ; 移栽自动回右下料位
OR 20.04  ; 移栽自动回左下料位
OR 20.05  ; 移栽自动回上料位
@PLS2(887) #0 #101 D610 D616  ; 移栽伺服自动加速度, 移栽伺服自动起动速度

### Section 自动报警

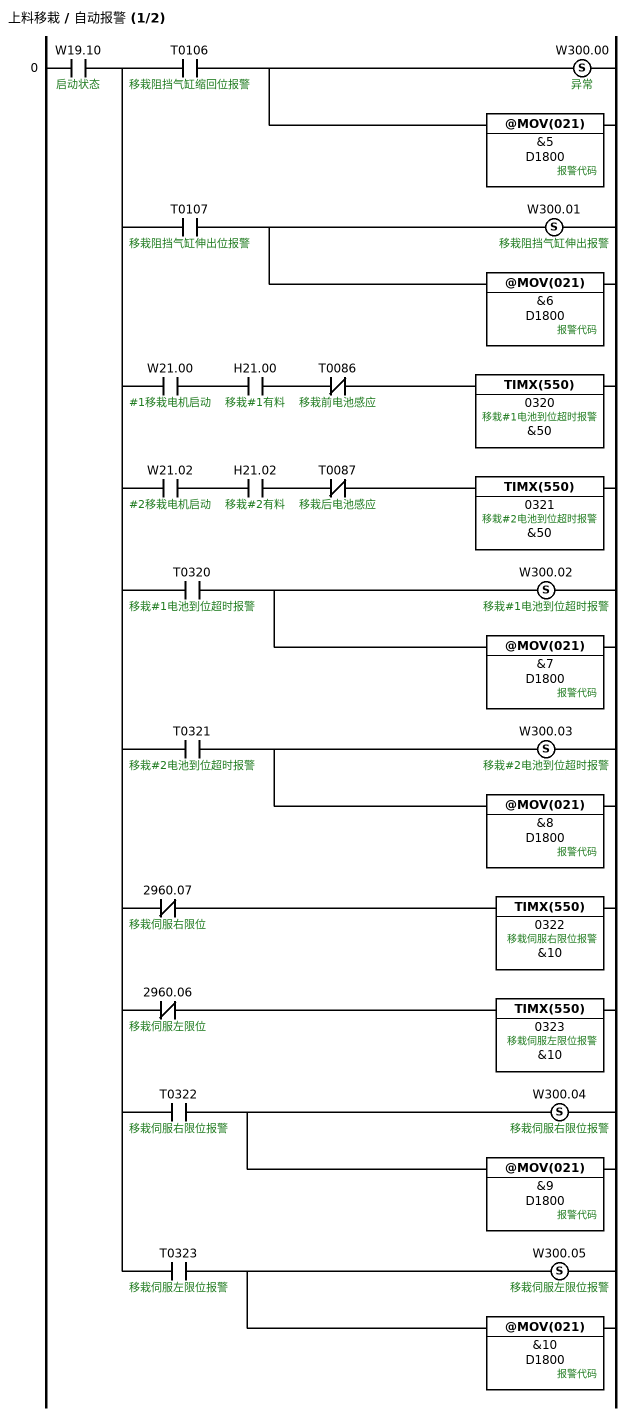
; rung 0
LD W19.10  ; 启动状态
OUT TR0
AND T0106  ; 移栽阻挡气缸缩回位报警
SET W300.00  ; 异常
@MOV(021) &5 D1800  ; 报警代码
LD TR0
AND T0107  ; 移栽阻挡气缸伸出位报警
SET W300.01  ; 移栽阻挡气缸伸出报警
@MOV(021) &6 D1800  ; 报警代码
LD TR0
AND W21.00  ; #1移栽电机启动
AND H21.00  ; 移栽#1有料
ANDNOT T0086  ; 移栽前电池感应
TIMX(550) 0320 &50  ; 移栽#1电池到位超时报警
LD TR0
AND W21.02  ; #2移栽电机启动
AND H21.02  ; 移栽#2有料
ANDNOT T0087  ; 移栽后电池感应
TIMX(550) 0321 &50  ; 移栽#2电池到位超时报警
LD TR0
AND T0320  ; 移栽#1电池到位超时报警
SET W300.02  ; 移栽#1电池到位超时报警
@MOV(021) &7 D1800  ; 报警代码
LD TR0
AND T0321  ; 移栽#2电池到位超时报警
SET W300.03  ; 移栽#2电池到位超时报警
@MOV(021) &8 D1800  ; 报警代码
LD TR0
ANDNOT 2960.07  ; 移栽伺服右限位
TIMX(550) 0322 &10  ; 移栽伺服右限位报警
LD TR0
ANDNOT 2960.06  ; 移栽伺服左限位
TIMX(550) 0323 &10  ; 移栽伺服左限位报警
LD TR0
AND T0322  ; 移栽伺服右限位报警
SET W300.04  ; 移栽伺服右限位报警
@MOV(021) &9 D1800  ; 报警代码
LD TR0
AND T0323  ; 移栽伺服左限位报警
SET W300.05  ; 移栽伺服左限位报警
@MOV(021) &10 D1800  ; 报警代码

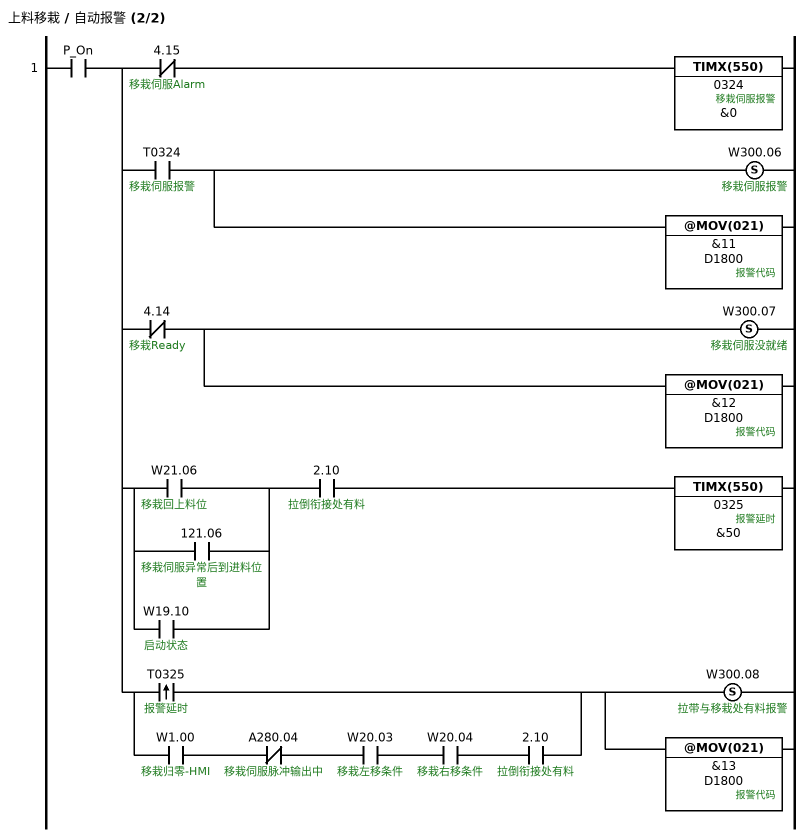
; rung 1
LD P_On
OUT TR0
ANDNOT 4.15  ; 移栽伺服Alarm
TIMX(550) 0324 &0  ; 移栽伺服报警
LD TR0
AND T0324  ; 移栽伺服报警
SET W300.06  ; 移栽伺服报警
@MOV(021) &11 D1800  ; 报警代码
LD TR0
ANDNOT 4.14  ; 移栽Ready
SET W300.07  ; 移栽伺服没就绪
@MOV(021) &12 D1800  ; 报警代码
LD TR0
LD W21.06  ; 移栽回上料位
OR 121.06  ; 移栽伺服异常后到进料位置
OR W19.10  ; 启动状态
ANDLD
AND 2.10  ; 拉倒衔接处有料
TIMX(550) 0325 &50  ; 报警延时
LD TR0
@LD T0325  ; 报警延时
LD W1.00  ; 移栽归零-HMI
ANDNOT A280.04  ; 移栽伺服脉冲输出中
AND W20.03  ; 移栽左移条件
AND W20.04  ; 移栽右移条件
AND 2.10  ; 拉倒衔接处有料
ORLD
ANDLD
SET W300.08  ; 拉带与移栽处有料报警
@MOV(021) &13 D1800  ; 报警代码

### Section 上料移栽复位

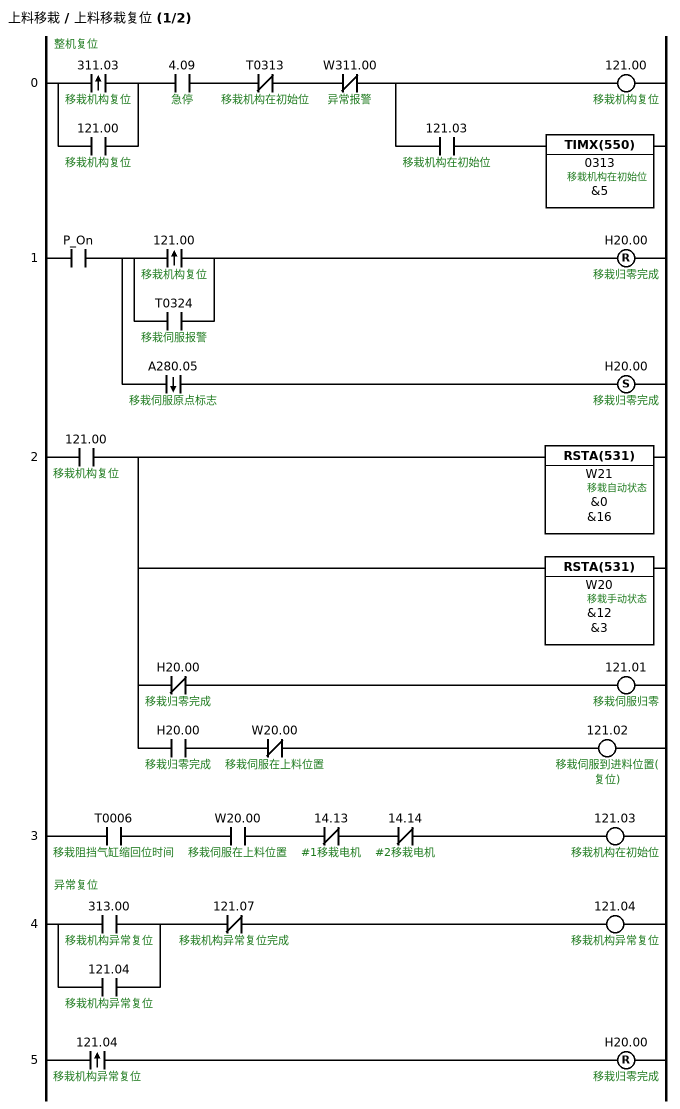
; rung 0: 整机复位
@LD 311.03  ; 移栽机构复位
OR 121.00  ; 移栽机构复位
AND 4.09  ; 急停
ANDNOT T0313  ; 移栽机构在初始位
ANDNOT W311.00  ; 异常报警
OUT 121.00  ; 移栽机构复位
AND 121.03  ; 移栽机构在初始位
TIMX(550) 0313 &5  ; 移栽机构在初始位
; rung 1
LD P_On
OUT TR0
@LD 121.00  ; 移栽机构复位
OR T0324  ; 移栽伺服报警
ANDLD
RSET H20.00  ; 移栽归零完成
LD TR0
%AND A280.05  ; 移栽伺服原点标志
SET H20.00  ; 移栽归零完成
; rung 2
LD 121.00  ; 移栽机构复位
OUT TR0
RSTA(531) W21 &0 &16  ; 移栽自动状态
RSTA(531) W20 &12 &3  ; 移栽手动状态
ANDNOT H20.00  ; 移栽归零完成
OUT 121.01  ; 移栽伺服归零
LD TR0
AND H20.00  ; 移栽归零完成
ANDNOT W20.00  ; 移栽伺服在上料位置
OUT 121.02  ; 移栽伺服到进料位置(复位)
; rung 3
LD T0006  ; 移栽阻挡气缸缩回位时间
AND W20.00  ; 移栽伺服在上料位置
ANDNOT 14.13  ; #1移栽电机
ANDNOT 14.14  ; #2移栽电机
OUT 121.03  ; 移栽机构在初始位
; rung 4: 异常复位
LD 313.00  ; 移栽机构异常复位
OR 121.04  ; 移栽机构异常复位
ANDNOT 121.07  ; 移栽机构异常复位完成
OUT 121.04  ; 移栽机构异常复位
; rung 5
@LD 121.04  ; 移栽机构异常复位
RSET H20.00  ; 移栽归零完成

